PROGRAM PRG_CaseErector

(*----------------------------------------------NOWE Wejściowe ------------------------------------------*)
VAR_INPUT
	eMachineMode							: E_LineMachineMode; 		// Machine mode
	eMachineCommand							: E_LineMachineCommand; 	// Command from top level state program
END_VAR
(*----------------------------------------------NOWE Wyjściowe ------------------------------------------*)
VAR_OUTPUT
	eMachineState							: E_CaseErectorMachineState;
  	bError									: BOOL;
END_VAR
(*----------------------------------------------NOWE Wewnętrzne ------------------------------------------*)
VAR
	// INPUTS
	bIn1									: BOOL;
	// OUTPUTS
	bOut1									: BOOL;	
	// Local
	iStateIdle								: INT;
	iStepStarting							: INT;
	iStateStoping							: INT;
	iStateAborting							: INT;	
	fbPower 								:MC_Power;
	fbMove	 								:MC_MoveAbsolute;
	fbJog 									:MC_Jog;
	fbReset 								:MC_Reset;	
	fbStop									:MC_Stop;
	//fbBeltInverter							:FB_MX2;
	arrErrorTable							:ARRAY[0..1000] OF UDINT;
	arrError								:ARRAY[0..1000] OF BOOL;
	tonAxesReady							:TON;
	tonAxesError							:TON;
	fbBeltInverter							:FB_INV003_MX2_ECT;
	ftSAFETY_PermissionSS1					:F_TRIG;
	ftSAFETY_PermissionSS2					:F_TRIG;
	
END_VAR
(*----------------------------------------------Koniec nowego dopisanego -------------------------------*)

ACTION Act_ButtonsLight:
IF  (gvl_hmi.A_Start=TRUE  THEN GVL_IO.K1K5:=FALSE; GVL_IO.K1K7:=TRUE; ; END_IF
IF gvl_hmi.A_Stop=TRUE THEN GVL_IO.K1K5:=TRUE; GVL_IO.K1K7:=FALSE;  END_IF
GVL_HMI.A_Start:=gvl_Io.b1K1;
GVL_HMI.A_Stop:=GVL_IO.b1K3;
END_ACTION

ACTION Act_CaseCycle:

END_ACTION

ACTION Act_Error:

END_ACTION

ACTION Act_FBsCall:
//Servo Axis Fb`s
	
fbPower(
	Axis:=GVL_AXIS.stAxis1 , 
	Enable:=, 
	Enable_Positive:=GVL_AXIS.bEnable , 
	Enable_Negative:=GVL_AXIS.bEnable , 
	Override:=100.0 , 
	BufferMode:= , 
	Options:= , 
	Status=> , 
	Busy=> , 
	Active=> , 
	Error=> arrError[0], 
	ErrorID=>arrErrorTable[0] );

fbReset(
	Axis:= GVL_AXIS.stAxis1, 
	Execute:= , 
	Done=> , 
	Busy=> , 
	Error=>	arrError[1] , 
	ErrorID=>arrErrorTable[1] );
		
fbJog(
	Axis:= GVL_AXIS.stAxis1, 
	JogForward:= bJog_B , 
	JogBackwards:=bJog_F , 
	Mode:= , 
	Position:= , 
	Velocity:= GVL_HMI.J_VelK, 
	Acceleration:= , 
	Deceleration:= , 
	Jerk:= , 
	Done=> , 
	Busy=> , 
	Active=> , 
	CommandAborted=> , 
	Error=> arrError[2] , 
	ErrorID=>arrErrorTable[2] );
	
fbMove(
	Axis:=GVL_AXIS.stAxis1 , 
	Execute:= , 
	Position:= , 
	Velocity:= , 
	Acceleration:= , 
	Deceleration:= , 
	Jerk:= , 
	BufferMode:= , 
	Options:= , 
	Done=> , 
	Busy=> , 
	Active=> , 
	CommandAborted=> , 
	Error=>arrError[3] , 
	ErrorID=>arrErrorTable[3]
 );
 fbStop(
	Axis:=GVL_AXIS.stAxis1 , 
	Execute:= , 
	Deceleration:= , 
	Jerk:= , 
	Options:= , 
	Done=> , 
	Busy=> , 
	Active=> , 
	CommandAborted=> , 
	Error=> arrError[4] , 
	ErrorID=>arrErrorTable[4] );
	//Inverters fb`s nie używany 
(*fbBeltInverter
	(w_Status:=GVL_Omron.wOmron_1_Status,
	ui_CzestotliwoscI:=F1_FQ,
	b_CCW:=F1_CW, 
	b_CW:=F1_CCW, 
	b_Reset:=F_Reset,		
	w_ControlW=>GVL_Omron.wOmron_1_Control,
 	ui_CzestotliwoscO=>GVL_Omron.iOmron_1_SeVelo,);
*)	

fbBeltInverter(
	Output_Frequency_Monitor:= , 
	During_Rev:= , 
	Enable:= , 
	Fwd:= , 
	Rev:= , 
	Fault_Reset:= , 
	Frequency_in:= , 
	Acceleration:= , 
	Deceleration:= , 
	ENO=> , 
	Frequency_out=>GVL_Omron.iOmron_1_SeVelo , 
	During_Fwd=> , 
	Fault=>arrError[5], 
	Warning=> , 
	Remote=> , 
	Freq_Match=> , 
	Connection_Error=> , 
	Command:=GVL_Omron.wOmron_1_Status , 
	Frequency_Reference:=GVL_Omron.iOmron_1_ActVelo , 
	F002_1st_Acceleration:=GVL_Omron.iOmronErectorAcc , 
	F003_1st_Deceleration:=GVL_Omron.iOmronErectorDcc , 
	Status:=GVL_Omron.wOmron_1_Status);
END_ACTION

ACTION Act_IOLinkRequest:
//załączenie kanału io-link Kanał 1 
		GVL_IO.IOLinkCh1T:=TRUE;
END_ACTION

ACTION Act_Magazine:
K_Magazyn(
	bStop:=GVL_IO.b1K3 AND GVL_HMI.bAuto,
	xPodjedz:=GVL_IO.b1K1, 
	xWydajKarton:=, 
	xKartonPobrany:=, 
	xCzPodjazd:=, 
	xCzTrzymacz2:=, 
	xCzTrzymacz1:=GVL_IO.bCzujnik_Trzymacz1, 
	xSilPodpych=>GVL_IO.K1K4, 
	xSilTrzymacz1=>GVL_IO.K1K1, 
	xSilTrzymacz2=>GVL_IO.K1K3, 
	xWydalemKarton=>, 
	xBlad=> );
END_ACTION

ACTION Act_ModeAutomatic:
// State Machine

CASE eMachineState OF

	E_MachineState.eIdle:
		
	
		// ====================================================
		// There should be main code
		// i.e. CASE iStepInit OF	
		// ====================================================
		// Allow for stop only if conditions are true - in this step we can wait without an error

		
		IF TRUE (* condition *) THEN
			eMachineState 						:= E_MachineState.eStopped;
		END_IF
		
		IF bError THEN
			eMachineState 						:= E_MachineState.eError;
		END_IF
		
	E_MachineState.eStopping:
		
		
		CASE iStateStoping OF
			0:
				
			10:
			
			20:
				
		END_CASE
		IF iStateStoping = 20 (* condition *) THEN
			eMachineState 						:= E_MachineState.eStopped;
			iStateStoping 						:= 0;
		END_IF		
	
	E_MachineState.eStopped:
		
	
		
		IF eMachineCommand = E_MachineCommand.eRun THEN
			eMachineState 						:= E_MachineState.eStarting;
		END_IF
		
		IF eMachineCommand = E_MachineCommand.eRestart THEN
			GVL_MachineMaintenance.eCommand		:= E_MachineCommand.eStop;
			eMachineState 						:= E_MachineState.eRestarting;
		END_IF			
				
		IF bError THEN
			eMachineState 						:= E_MachineState.eError;
		END_IF

	E_MachineState.eStarting:
	

		CASE iStepStarting OF
			0:		
				fbPower.Enable:=TRUE;
				
				IF tonAxesReady.Q THEN
					iStepStarting := iStepStarting + 10;
				ELSIF tonAxesError.Q THEN
					bError := TRUE;
				END_IF
			
			10:
			
				IF (*Warunki startu automatu*)  THEN
					iStepStarting := iStepStarting + 20;		
				ELSE
					bError := TRUE;
					iStepStarting := iStepStarting + 10;
				END_IF
				
			20:
			
		
				
			END_CASE 
	
		IF iStepStarting = 20 AND (*Kartoniarka READY*) THEN
			eMachineState 						:= E_MachineState.eRunning;
			iStepStarting 						:= 0;
		END_IF
		
			
		
	E_MachineState.eRunning:
		

		// ====================================================
		// There should be main code
		// i.e. CASE iStepAuto OF
		// ====================================================
		IF eMachineCommand = E_MachineCommand.eStop OR bError THEN
			eMachineState 						:= E_MachineState.eStopping;
		END_IF

	E_MachineState.eAborting:

		// Stop and reset everything - usually SAFETY function
		CASE iStateAborting OF
			0:
				IF  ftSAFETY_PermissionSS1.Q  OR  ftSAFETY_PermissionSS2.Q   (*warunek wykonania zatrzymania *) THEN
					iStateAborting := iStateAborting +10;
				END_IF
			10:
				
						fbMove.Execute:= FALSE;
						fbStop.Execute:= TRUE;
						
						IF fbStop.Done THEN
							fbStop.Execute:= FALSE;
							iStateAborting := iStateAborting +10;	
						END_IF
				
			20:
						fbPower.Enable:=FALSE;
					IF NOT fbPower.Status THEN 
						iStateAborting := iStateAborting + 10;
					END_IF
			30:
			
					
				
		END_CASE
	
		IF iStateAborting = 30 THEN
			eMachineState 						:= E_MachineState.eAborted;
			iStateAborting						:= 0;
		END_IF		
		
	E_MachineState.eAborted:

					
		IF eMachineCommand = E_MachineCommand.eReset THEN
			eMachineState 						:= E_MachineState.eReseting;
		END_IF
		
		IF bError THEN
			eMachineState 						:= E_MachineState.eError;
		END_IF

	E_MachineState.eError:

		// ====================================================
		// Two types of error:
		// 1. 'Small/soft' Error - fix a problem and go to stop
		// 2. 'Serious/hard' Error - there is a need of restart everything, if there is a sequence - reset it too - fix a problem and go to init
		// ====================================================

	
	
		IF eMachineCommand = E_MachineCommand.eReset THEN
			eMachineState 						:= E_MachineState.eReseting;
		END_IF
		
		IF eMachineCommand = E_MachineCommand.eRestart THEN
			eMachineState 						:= E_MachineState.eRestarting;
		END_IF

	E_MachineState.eReseting:

		// ====================================================
		//'Small/soft' Error - fix a problem and go to stop
		// Reset drives only when it is necessary
		// ====================================================
		// Check if axis errors cleared
	
		IF fbPower.Error	THEN
			fbReset.Execute := TRUE;
		ELSIF fbBeltInverter.Fault THEN
			fbBeltInverter.Fault_Reset:=TRUE;
		ELSIF fbPower.Error OR fbJog.Error OR fbMove.Error OR fbStop.Error OR GVL_AXIS.stAxis1.Status.Error THEN
			fbReset.Execute:=TRUE;
			
	END_IF

	
		IF NOT tonAxesError.Q  THEN
			fbReset.Execute := FALSE;
			fbBeltInverter.Fault_Reset:=FALSE;
		END_IF
				
		// Blad bloku resetowania lub zakonczylismy kasowanie bledu osi, ale os jest nadal w bledzie, np. nie usunieta usterka - idz do kroku bledu
		IF bError (*(stAxis.stAxisDiagOutputs.Error OR (stAxis.stAxisDiagOutputs.Done AND stAxis.bAxisError)) *) THEN
			eMachineState  						:= E_MachineState.eError;
		END_IF
		
	E_MachineState.eRestarting:

		// ====================================================
		// 'Serious/hard' Error - there is a need of restart everything, if there is a sequence - reset it too - fix a problem and go to init
		// Reset drives only when it is necessary
		// ====================================================
		// Check if axis errors cleared
		bError := FALSE;
		
		IF TRUE (*NOT bAxisError AND NOT other errors *) THEN
			eMachineState  						:= E_MachineState.eIdle;
		END_IF
				
		// Blad bloku resetowania lub zakonczylismy kasowanie bledu osi, ale os jest nadal w bledzie, np. nie usunieta usterka - idz do kroku bledu
		IF bError (*(stAxis.stAxisDiagOutputs.Error OR (stAxis.stAxisDiagOutputs.Done AND stAxis.bAxisError)) *) THEN
			eMachineState  						:= E_MachineState.eError;
		END_IF
		
END_CASE

ftSAFETY_PermissionSS1(CLK:=GVL_SafetyFrom_RT2.bSAFETY_PermissionSS1);
ftSAFETY_PermissionSS2(CLK:=GVL_SafetyFrom_RT2.bSAFETY_PermissionSS2);
END_ACTION

ACTION Act_ModeManual:

END_ACTION

ACTION Act_Monitoring:
tonAxesReady(PT:=T#200MS);
tonAxesReady.IN:=fbPower.Active;

tonAxesError(PT:=T#200MS);
tonAxesError.IN:=arrError[0] OR arrError[1] OR arrError[2]  OR arrError[5]
							 OR arrError[3] OR arrError[4];
END_ACTION

END_PROGRAM

(* stored: Version 1.1.0.1, ProductVersion 3.1.4022.12
   POU PRG_CaseErector: Id {787febfa-fe21-4eba-bbd9-2fbeb26b9e96}, SpecialFunc None
   Action Act_ButtonsLight: Id {976c460d-ce54-4d95-a684-d06828d38226}
   Action Act_CaseCycle: Id {057b89b8-516c-4a83-bfcc-0cb20ed81027}
   Action Act_Error: Id {d847853c-0914-4802-bce7-bd5b5e3321aa}
   Action Act_FBsCall: Id {9fbcae2a-f886-48dc-a8fd-b42be9c44f4d}
   Action Act_IOLinkRequest: Id {d80c0f49-d643-4e27-9599-7ce7ea085bdf}
   Action Act_Magazine: Id {7f1f6fa3-4a22-4cb2-b4c0-4e2ecc8ef5c4}
   Action Act_ModeAutomatic: Id {f4ca6b94-7366-4b9f-a3a5-13513218a207}
   Action Act_ModeManual: Id {de63055e-42c1-4b42-bc45-31e1849e99a1}
   Action Act_Monitoring: Id {32ce7dfd-1d1b-42ec-9e3a-a2f9429ed76b} *)
